TYPE
    U_FourByteDigitalControlInput :
    UNION
        uUint  : UINT;
        aBytes : ARRAY[0..3] OF BYTE;
    END_UNION
END_TYPE

(* stored: Version 1.1.0.1, ProductVersion 3.1.4024.12
   DUT U_FourByteDigitalControlInput: Id {f8024516-d16f-42a9-b023-735c97c4a13d} *)
